{attribute 'GeneratedUsingTerminal: EP9224-0037-0017'}
{attribute addProperty BoxType "EP9224-0037-0017"}
{attribute addProperty Id "Device_StatusAT %I*Device_Status_033C68E911Current_UsAT %I*INT2Current_UpAT %I*INT2Voltage_UsAT %I*INT2Voltage_UpAT %I*INT2TemperatureAT %I*INT2"}
{attribute addProperty CRC "202813344"}
{attribute addProperty Size "21"}
TYPE DPO_Inputs_Device_0C16AFA0 :
STRUCT
	{attribute addProperty Name "Device_Status"}
	Device_Status AT %I* : Device_Status_033C68E9;
	{attribute addProperty Name "Current_Us"}
	Current_Us AT %I* : INT;
	{attribute addProperty Name "Current_Up"}
	Current_Up AT %I* : INT;
	{attribute addProperty Name "Voltage_Us"}
	Voltage_Us AT %I* : INT;
	{attribute addProperty Name "Voltage_Up"}
	Voltage_Up AT %I* : INT;
	{attribute addProperty Name "Temperature"}
	Temperature AT %I* : INT;
END_STRUCT
END_TYPE

(* stored: Version 1.2.0.0, ProductVersion 3.1.4024.9
   DUT DPO_Inputs_Device_0C16AFA0: Id {80685ca0-25f3-4e65-8006-1faa1c722e6d} *)
